(* Logix 5000 project; controller LDSDKdemo_simpleEx_L85E_v36 1756-L85E rev 38.11; software revision 38.01 *)

TASK T00_Task (continuous, watchdog 500 ms) : P00_Program

MODULES
   Local : 1756-L85E (ICP 0, rev 38.11)
END_MODULES

VAR_GLOBAL   (* controller tags *)
   area_comparison_result1 : BOOL;
   box_length : SINT;
   box_width : DINT;
   compareValue_for_box_Area : DINT;
END_VAR

PROGRAM P00_Program   (* main routine R00_MainRoutine *)
VAR
   box_area : LINT;
END_VAR

ROUTINE R00_MainRoutine   (* ladder *)
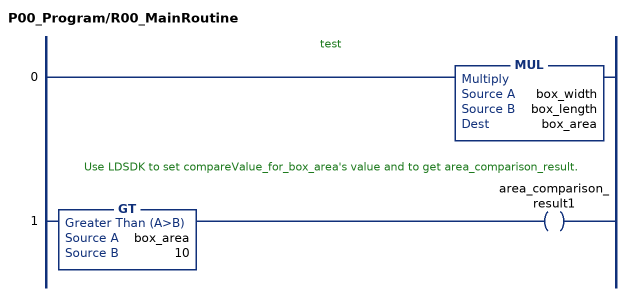
   // test
   0: MUL(box_width,box_length,box_area);
   // Use LDSDK to set compareValue_for_box_area's value and to get area_comparison_result.
   1: GT(box_area,10)OTE(area_comparison_result1);
END_ROUTINE
END_PROGRAM
